// TIA Portal V18 export
TYPE "PLCtoMES_Common"
// stored: IsFailsafeCompliant false
   STRUCT
      "P-HeartBeat" : Bool;   // MES心跳信号，频率5S，PLC10S延迟判定报警
      "P-AtPreStop" : Bool;   // 工件预停开始放行，到工件到位，算物流时间
      "P-AtPro" : Bool;   // 托盘在位标志位，托盘到位后PLC置位，托盘离开后PLC复位
      "P-AtWork" : Bool;   // 循环状态标志位，MES允许加工后由PLC置位，循环结束后由PLC复位
      "P-EquipStatus" : Byte;   // 关机：9急停：10异常停机：20换刀：25空循环：30其它：35通过模式：37非自动模式：40循环停止：60特殊模式：70堵料：83待料：86等待：90生产中：100
      "P-EquipMode" : Byte;   // 设备循环模式（1-手动，2自动，3旁通，4空循环 -5-标定）
      "P-BuffQTY" : Array[1..10] of DInt;   // 工段/工位缓存数量
      Reserve : Array[1..155] of Byte;   // 设备状态字预留
   END_STRUCT;
END_TYPE
